TYPE T_PIEZO_DINT :
STRUCT
	nValue:	DINT;
END_STRUCT
END_TYPE

(* stored: Version 1.1.0.1, ProductVersion 3.1.4022.16
   DUT T_PIEZO_DINT: Id {e593f3da-de92-42fc-aac0-0f07efb3b6ed} *)
